// TIA Portal V15 export
// export: Created 2018-05-29T12:25:38.1552518Z, ExportSetting WithDefaults, DisplayName Totally Integrated Automation Portal, DisplayVersion V15, DisplayName STEP 7 Professional, DisplayVersion V15, DisplayName WinCC Professional, DisplayVersion V15, DisplayName TIA Portal Openness, DisplayVersion V15
FUNCTION "phase_2_fc" : Void   // FC1, STL
TITLE = _fc
{ S7_Optimized_Access := 'TRUE' }
VERSION : 0.1
// Second instance of fds_example test
// stored: AutoNumber true, UDAEnableTagReadback false
BEGIN

NETWORK
TITLE = Main
// comment: Second instance of fds_example


// Call the EM FB with the corresponding DB instance
      CALL  "phase_example", "phase_2"
      ( scantime                := ,
        Bool1                   := ,
        Bool2                   := ,
        EM_I_OUT_ID             := #"",
        Some_Dyn_EM_ID          := ,
        DB_NO                   := ,
        XV003_OPN               := #"XV301.QOPEN",
        XV003_CLS               := #"XV301.QCLOSE",
        XV003_MERR              := #"XV301.QMON_ERR",
        XV004_OPN               := #"XV401.QOPEN",
        XV004_CLS               := #"XV401.QCLOSE",
        XV004_MERR              := #"XV401.QMON_ERR",
        XV005_OPN               := #"XV501.QOPEN",
        XV005_CLS               := #"XV501.QCLOSE",
        XV005_MERR              := #"XV501.QMON_ERR",
        P001_RUN                := #"P101.QRUN",
        P001_STOP               := #"P101.QSTOP",
        P001_MERR               := #"P101.QMON_ERR",
        P001_MPS                := #"P101.QMPS",
        P002_RUN                := #"P201.QRUN",
        P002_STOP               := #"P201.QSTOP",
        P002_MERR               := #"P201.QMON_ERR",
        P002_MPS                := #"P201.QMPS",
        EM_I_OUT_OWN            := ,
        EM_I_OUT_STA            := ,
        EM_I_OUT_ERR            := ,
        EM_I_OUT_ERRNO          := ,
        EM_I_OUT_ACTIV          := ,
        EM_I_OUT_LT             := ,
        EM_I_OUT_PT             := ,
        LT001_PV                := #"LT101.QfVal",
        LT001_AHH               := #"LT101.LIM_Qb01",
        LT001_AH                := #"LT101.LIM_Qb02",
        LT001_AL                := #"LT101.LIM_Qb03",
        LT001_ALL               := #"LT101.LIM_Qb04",
        LT001_ERR               := #"LT101.QERR",
        LT002_PV                := #"LT201.QfVal",
        LT002_AHH               := #"LT201.LIM_Qb01",
        LT002_AH                := #"LT201.LIM_Qb02",
        LT002_AL                := #"LT201.LIM_Qb03",
        LT002_ALL               := #"LT201.LIM_Qb04",
        LT002_ERR               := #"LT201.QERR",
        FIC001_PV               := #"FIC101.PV",
        FIC001_ERR              := #"FIC101.QERR",
        Some_Dyn_EM_OWN         := ,
        Some_Dyn_EM_STA         := ,
        Some_Dyn_EM_ERR         := ,
        Some_Dyn_EM_ERRNO       := ,
        Some_Dyn_EM_ACTIV       := ,
        Some_Dyn_EM_LT          := ,
        Some_Dyn_EM_PT          := ,
        XV008_OPN               := ,
        XV008_CLS               := ,
        XV008_MERR              := ,
        phase_id                := ,
        state                   := ,
        stepnumber              := ,
        message                 := ,
        button_1_text           := ,
        button_2_text           := ,
        button_3_text           := ,
        button_1_visible        := ,
        button_2_visible        := ,
        button_3_visible        := ,
        button_reverse          := ,
        state_idle              := ,
        state_running           := ,
        state_complete          := ,
        state_pausing           := ,
        state_paused            := ,
        state_holding           := ,
        state_held              := ,
        state_restarting        := ,
        state_stopping          := ,
        state_stopped           := ,
        state_aborting          := ,
        state_aborted           := ,
        enable_start            := ,
        enable_stop             := ,
        enable_hold             := ,
        enable_restart          := ,
        enable_abort            := ,
        enable_reset            := ,
        enable_pause            := ,
        enable_resume           := ,
        enable_auto             := ,
        enable_man              := ,
        enable_byte             := ,
        auto                    := ,
        steptime_s              := ,
        steptime_m              := ,
        steptime_h              := ,
        MSG_no01                := ,
        MSG_no02                := ,
        MSG_no03                := ,
        MSG_no04                := ,
        MSG_no05                := ,
        MSG_no06                := ,
        MSG_no07                := ,
        MSG_no08                := ,
        MSG_no09                := ,
        MSG_no10                := ,
        Destination             := ,
        setpoint                := ,
        some_bool_out           := ,
        XV003_CMD               := #"XV301.AUT_OP",
        XV004_CMD               := #"XV401.AUT_OP",
        XV005_CMD               := #"XV501.AUT_OP",
        P001_ON                 := #"P101.AUTO_ON",
        P001_AUT                := #"P101.L_AUT",
        P002_ON                 := #"P201.AUTO_ON",
        P002_AUT                := #"P201.L_AUT",
        EM_I_OUT_REQ            := ,
        EM_I_OUT_CMD            := ,
        EM_I_OUT_P_SP           := ,
        FIC001_EXT              := #"FIC101.L_REMOTE",
        FIC001_SP               := #"FIC101.HMI_SP_INT",
        FIC001_AUT              := #"FIC101.L_AUT",
        FIC001_VAL_OUT          := #"FIC101.HMI_MAN",
        FIC001_SET_SP           := #"FIC101.Set_SP",
        FIC001_SET_OUT          := #"FIC101.Set_Output",
        Some_Dyn_EM_REQ         := ,
        Some_Dyn_EM_CMD         := ,
        Some_Dyn_EM_P_SP        := ,
        timer_dosing_pause      := ,
        timer_dosing_s          := ,
        timer_dosing_m          := ,
        timer_dosing_h          := ,
        timer_mixing_pause      := ,
        timer_mixing_s          := ,
        timer_mixing_m          := ,
        timer_mixing_h          := ,
        timer_circulation_pause := ,
        timer_circulation_s     := ,
        timer_circulation_m     := ,
        timer_circulation_h     := ,
        XV008_CMD               := ,
        plc_commands            := ,
        hmi_commands            := ,
        hmi_par_without_unit    := ,
        timesetting             := 
      );
END_FUNCTION
